// SIMATIC S7-200 project (STEP 7-Micro/WIN), CPU 224 UN REL 02.01

ORGANIZATION_BLOCK 主程序:OB1
TITLE=程序注释
BEGIN
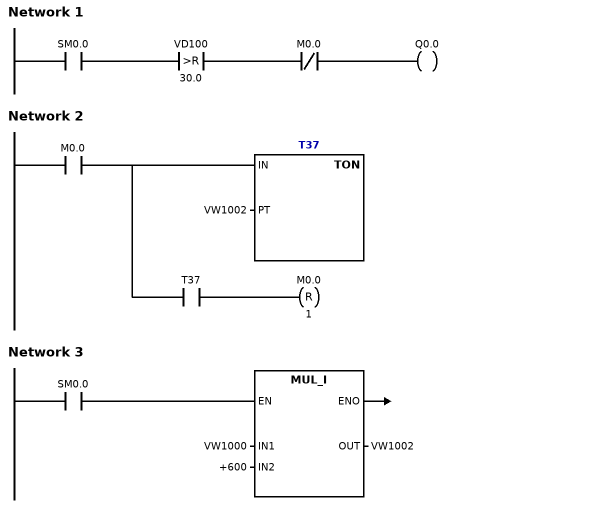
Network 1
LD     SM0.0
AR>    VD100, 30.0
AN     M0.0
=      Q0.0
Network 2
LD     M0.0
TON    T37, VW1002
A      T37
R      M0.0, 1
Network 3
// (network saved uncompiled; LAD cells follow)
// row 0: c0 -| |- SM0.0  c1 --  c2 [MUL_I EN:=power@row0, IN1:=VW1000, IN2:=+600, ENO=>power, OUT=>VW1002]  c3 ->
// row 1: c2 [box]
END_ORGANIZATION_BLOCK

SUBROUTINE_BLOCK SBR_0:SBR0
TITLE=子程序注释
BEGIN
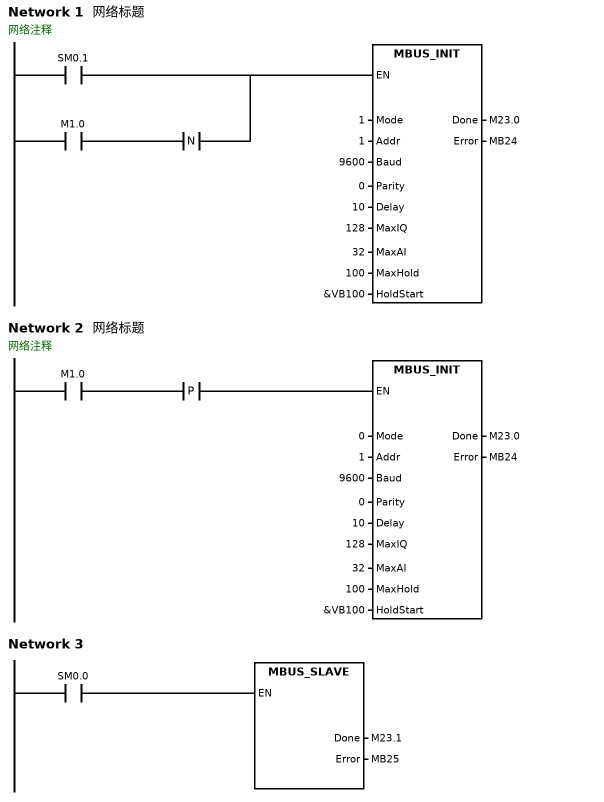
Network 1 // 网络标题
// 网络注释
LD     SM0.1
LD     M1.0
ED
OLD
CALL   MBUS_INIT:SBR2, 1, 1, 9600, 0, 10, 128, 32, 100, &VB100, M23.0, MB24
Network 2 // 网络标题
// 网络注释
LD     M1.0
EU
CALL   MBUS_INIT:SBR2, 0, 1, 9600, 0, 10, 128, 32, 100, &VB100, M23.0, MB24
Network 3
LD     SM0.0
CALL   MBUS_SLAVE:SBR3, M23.1, MB25
END_SUBROUTINE_BLOCK

// SBR1: protected block, not included

// SBR2: protected block, not included

// SBR3: protected block, not included

// SBR4: protected block, not included
